INTERFACE ITcMessage_Ext

PROPERTY LoggerLevel : TcEventSeverity
GET
END_GET
SET
END_SET
END_PROPERTY

METHOD Send : BOOL
VAR_INPUT
	eventType : Tc3_EventLogger.TcEventEntry;
	args : STRING(255);
END_VAR
END_METHOD

END_INTERFACE

(* stored: Version 1.1.0.1, ProductVersion 3.1.4024.11
   Itf ITcMessage_Ext: Id {ecc02940-e99f-4b59-aa27-20f74ac0a53f}
   Property LoggerLevel: Id {0e41f927-4626-478b-91df-4414fd23a8d2}
   Get Get: Id {5d3ace24-bef4-4c37-bf66-65ddbe71722a}
   Set Set: Id {324ec054-699b-48a8-8e04-7f635f59a639}
   Method Send: Id {974ef709-63a5-449e-b808-feae03cbbc39} *)
